SUBAPPLICATION logiBUS_PI_IDA_OPC (* logiBUS_PI_IDA (Puls-Eingang) auf VT-Zahlenfelder (Zaehler roh + Frequenz Hz, je eigene CNumberVariable) + Bargraph (Frequenz) + OPC-UA (Zaehler DWORD + Frequenz REAL, generisch, ein Kanal) *)
  (* Standard: 61499-2; Description: Copyright (c) 2026 Meisterschulen am Ostbahnhof This program and the accompanying materials are made available under the terms of the Eclipse Public License 2.0 which is available at https://www.eclipse.org/legal/epl-2.0/ SPDX-License-Identifier: EPL-2.0 *)
  (* Version 1.0, 2026-08-30, Franz Höpfinger, Meisterschulen am Ostbahnhof, initial API and implementation and/or initial documentation *)
  PACKAGE MyLib::sys;
  IMPORT isobus::UT::Q::const::IDs::ID_NULL;
  IMPORT logiBUS::io::PI::logiBUS_PI;
  IMPORT logiBUS::io::PI::logiBUS_PI_S;
  IMPORT logiBUS::utils::conversion::phys::NumericObjectPool_S;
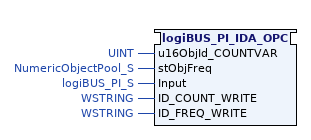
  VAR_INPUT
    u16ObjId_COUNTVAR : UINT := ID_NULL; (* Object ID CNumberVariable (roher Zaehlerstand, unbegrenzt wachsend, Scale=1 im VT-Pool) *)
    stObjFreq : logiBUS::utils::conversion::phys::NumericObjectPool_S := (u16ObjId := ID_NULL, r32Scale := 1.0, i32Offset := 0, u8Decimals := 0); (* Object ID + Scale/Offset/Decimals CNumberVariable (Frequenz Hz, eigene, unabhaengige CNumberVariable - keine Reskalierung des Zaehlers) *)
    Input : logiBUS::io::PI::logiBUS_PI_S := logiBUS_PI::Invalid; (* Identify the Input PulseInput_I1..I8 *)
    ID_COUNT_WRITE : WSTRING; (* Zaehler-Ruckmelde-Adresse (DWORD, roh, ACTION=PUBLISH) *)
    ID_FREQ_WRITE : WSTRING; (* Frequenz-Ruckmelde-Adresse (REAL Hz, ACTION=PUBLISH) *)
  END_VAR
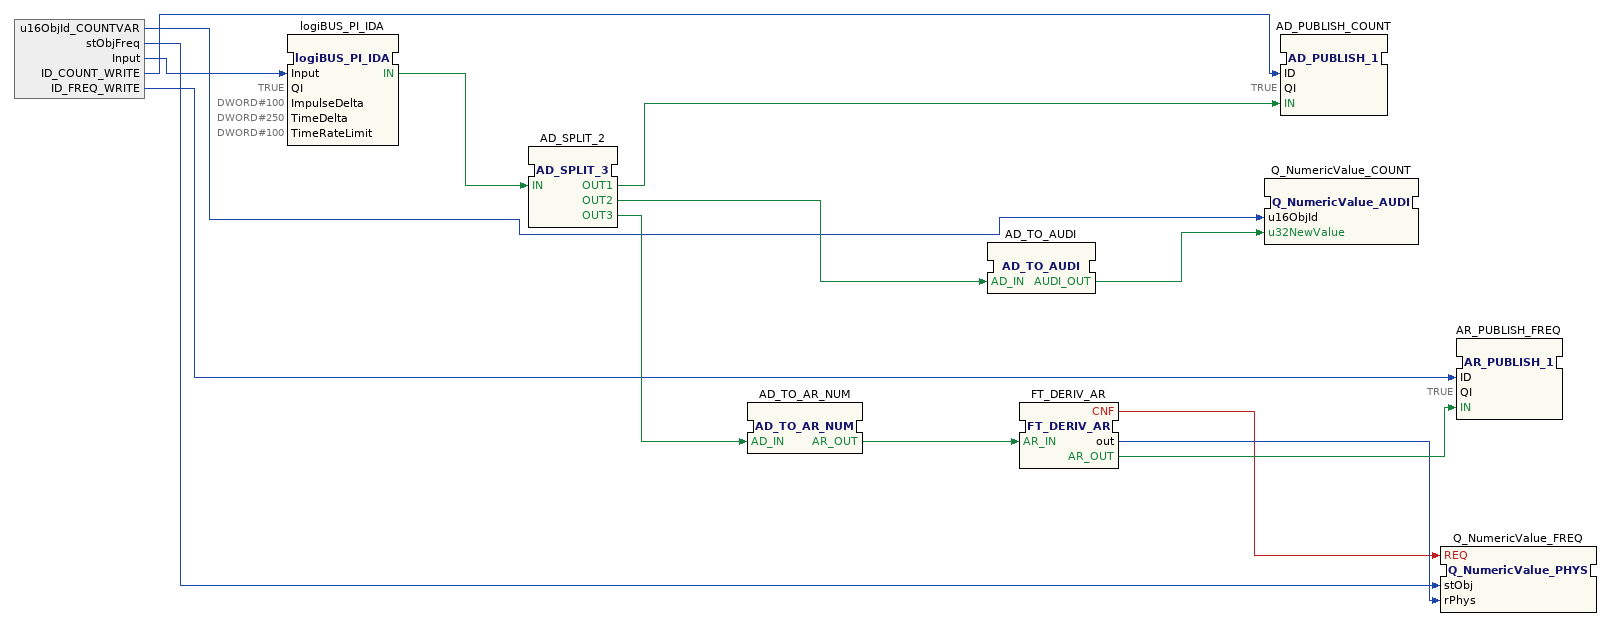
  FBS
    logiBUS_PI_IDA : logiBUS::io::PI::logiBUS_PI_IDA(QI := TRUE, ImpulseDelta := DWORD#100, TimeDelta := DWORD#250, TimeRateLimit := DWORD#100);
    AD_SPLIT_2 : adapter::events::unidirectional::AD_SPLIT_3;
    AD_PUBLISH_COUNT : adapter::net::AD_PUBLISH_1(QI := TRUE);
    AD_TO_AUDI : adapter::conversion::unidirectional::AD_TO_AUDI;
    Q_NumericValue_COUNT : isobus::UT::Q::Q_NumericValue_AUDI;
    AD_TO_AR_NUM : adapter::conversion::unidirectional::AD_TO_AR_NUM;
    FT_DERIV_AR : OSCAT_adapter::Control::FT_DERIV_AR;
    AR_PUBLISH_FREQ : adapter::net::AR_PUBLISH_1(QI := TRUE);
    Q_NumericValue_FREQ : isobus::UT::Q::Q_NumericValue_PHYS;
  END_FBS
  EVENT_CONNECTIONS
    FT_DERIV_AR.CNF TO Q_NumericValue_FREQ.REQ;
  END_CONNECTIONS
  DATA_CONNECTIONS
    Input TO logiBUS_PI_IDA.Input;
    u16ObjId_COUNTVAR TO Q_NumericValue_COUNT.u16ObjId;
    stObjFreq TO Q_NumericValue_FREQ.stObj;
    ID_COUNT_WRITE TO AD_PUBLISH_COUNT.ID;
    ID_FREQ_WRITE TO AR_PUBLISH_FREQ.ID;
    FT_DERIV_AR.out TO Q_NumericValue_FREQ.rPhys;
  END_CONNECTIONS
  ADAPTER_CONNECTIONS
    logiBUS_PI_IDA.IN TO AD_SPLIT_2.IN;
    AD_SPLIT_2.OUT1 TO AD_PUBLISH_COUNT.IN;
    AD_SPLIT_2.OUT2 TO AD_TO_AUDI.AD_IN;
    AD_SPLIT_2.OUT3 TO AD_TO_AR_NUM.AD_IN;
    AD_TO_AUDI.AUDI_OUT TO Q_NumericValue_COUNT.u32NewValue;
    AD_TO_AR_NUM.AR_OUT TO FT_DERIV_AR.AR_IN;
    FT_DERIV_AR.AR_OUT TO AR_PUBLISH_FREQ.IN;
  END_CONNECTIONS
END_SUBAPPLICATION
